KUKA KRL data list: tipdress2.dat

&ACCESS RV1
&REL 33
&COMMENT TIPDRESS EXTERNAL GUN 2
DEFDAT  TIPDRESS2
;FOLD EXTERNAL DECLARATIONS;%{PE}%MKUKATPBASIS,%CEXT,%VCOMMON,%P
;FOLD GRIPPERTECH EXT
EXT  H50 (INT  :IN,INT  :IN,INT  :IN,GRP_TYP  :IN )
;ENDFOLD (GRIPPERTECH EXT)
;FOLD SPOTTECH EXT
EXT  USERSPOT (S_COMMAND  :IN,SPOT_TYPE  :IN )
;ENDFOLD (SPOTTECH EXT)
;FOLD BASISTECH EXT;%{PE}%MKUKATPBASIS,%CEXT,%VEXT,%P
EXT  BAS (BAS_COMMAND  :IN,REAL  :IN )
DECL INT SUCCESS
;ENDFOLD (BASISTECH EXT)
;FOLD USER EXT;%{E}%MKUKATPUSER,%CEXT,%VEXT,%P
;Make here your modifications
;ENDFOLD (USER EXT)
;ENDFOLD (EXTERNAL DECLERATIONS)
;FOLD USER EXT;%{}%V2.2.2,%MKUKATPUSER,%CEXT,%VEXT,%P
;Make here your modifications
DECL BOOL TIPKONTROLE
DECL INT ANSWER
DECL INT WAITTIME=5
;ENDFOLD
;ENDFOLD
DECL INT I

;******************************
;*     E6POS Declarations     *
;******************************

DECL E6POS XP10={X 1812.73999,Y -758.109497,Z 1603.28101,A -10.9368095,B 87.2611084,C -2.35136199,S 6,T 50,E1 0.0,E2 0.0,E3 0.0,E4 0.0,E5 0.0,E6 0.0}
DECL E6POS XP20={X -1662.00305,Y -1200.49304,Z 238.679993,A 92.3594437,B 77.6989288,C -175.853195,S 6,T 26,E1 -667.745789,E2 0.0,E3 0.0,E4 0.0,E5 0.0,E6 0.0}
DECL E6POS XBEFORETIPDRESS={X -1664.84497,Y -1195.28101,Z 131.821106,A 92.7083206,B 79.2879791,C -177.241806,S 6,T 26,E1 -667.74939,E2 0.0,E3 0.0,E4 0.0,E5 0.0,E6 0.0}
DECL E6POS XDRESS_POS={X -1664.83301,Y -1250.33301,Z 131.817993,A 92.7068863,B 79.2882233,C -177.243393,S 6,T 26,E1 -667.74762,E2 0.0,E3 0.0,E4 0.0,E5 0.0,E6 0.0}
DECL E6POS XAFTERTIPDRESS={X -1664.84497,Y -1195.28101,Z 131.821106,A 92.7083206,B 79.2879791,C -177.241806,S 6,T 26,E1 -667.74939,E2 0.0,E3 0.0,E4 0.0,E5 0.0,E6 0.0}
DECL E6POS XBEST_PRACKTICE={X -1662.02905,Y -1184.83496,Z 277.771301,A 92.3578873,B 77.6946869,C -175.853302,S 6,T 26,E1 -667.74762,E2 0.0,E3 0.0,E4 0.0,E5 0.0,E6 0.0}
DECL E6POS XP30={X -958.122009,Y 929.273499,Z 985.610474,A 92.0788727,B 72.5539932,C -179.8358,S 6,T 26,E1 -2887.17505,E2 0.0,E3 0.0,E4 0.0,E5 0.0,E6 0.0}

;******************************
;*      FDAT Declarations     *
;******************************

DECL FDAT FP10={TOOL_NO 14,BASE_NO 0,IPO_FRAME #BASE,TQ_STATE FALSE}
DECL FDAT FP20={TOOL_NO 1,BASE_NO 0,IPO_FRAME #BASE}
DECL FDAT FBEFORETIPDRESS={TOOL_NO 1,BASE_NO 0,IPO_FRAME #BASE}
DECL FDAT FDRESS_POS={TOOL_NO 1,BASE_NO 0,IPO_FRAME #BASE}
DECL FDAT FAFTERTIPDRESS={TOOL_NO 1,BASE_NO 0,IPO_FRAME #BASE}
DECL FDAT FBEST_PRACKTICE={TOOL_NO 1,BASE_NO 0,IPO_FRAME #BASE}
DECL FDAT FP30={TOOL_NO 1,BASE_NO 0,IPO_FRAME #BASE}

;******************************
;*  PDAT & LDAT Declarations  *
;******************************

DECL PDAT PH={VEL 100.0,ACC 100.0,APO_DIST 100.0}

DECL E6POS XBEST_PRAKTISCH={X 1813.98499,Y -755.127197,Z 1603.28101,A -10.8495102,B 87.2611771,C -2.35826492,S 6,T 50,E1 0.0,E2 0.0,E3 0.0,E4 0.0,E5 0.0,E6 0.0}
DECL SPOT_SUGG_T LAST_SPOT={GUN[] "1                       ",RETR_CMD[] "#OPN                    ",CHOISE[] "#FIRST                  ",CLO_TM[] "0                       ",PGNO1[] "1                       ",PRESS1[] "0                       ",PGNO2[] "1                       ",PRESS2[] "0                       ",SPOT_PARAMS[] "SDAT3                   "}
DECL BASIS_SUGG_T LAST_BASIS={POINT1[] "Best_Praktisch          ",POINT2[] "Best_Praktisch          ",CP_PARAMS[] "CPDAT0                  ",PTP_PARAMS[] "H                       ",CONT[] "                        ",CP_VEL[] "2.0                     ",PTP_VEL[] "100                     ",SPL_NAME[] "S0                      "}
DECL FDAT FBest_Praktisch={TOOL_NO 14,BASE_NO 0,IPO_FRAME #BASE,POINT2[] " ",TQ_STATE FALSE}
DECL PDAT PPDAT1={VEL 100.0,ACC 100.0,APO_DIST 100.0}
DECL E6POS XBest_Praktice={X -1662.07202,Y -1184.76196,Z 277.795013,A 92.3631592,B 77.6921463,C -175.8461,S 6,T 26,E1 -667.74762,E2 0.0,E3 0.0,E4 0.0,E5 0.0,E6 0.0}
DECL FDAT FBest_Praktice={TOOL_NO 1,BASE_NO 0,IPO_FRAME #BASE,POINT2[] " "}
DECL E6POS XP21={X -929.55603,Y -159.533905,Z 748.283386,A 92.0804672,B 72.5703812,C -179.830597,S 6,T 26,E1 -2646.86792,E2 0.0,E3 0.0,E4 0.0,E5 0.0,E6 0.0}
DECL FDAT FP21={TOOL_NO 1,BASE_NO 0,IPO_FRAME #BASE}
DECL E6POS XP31={X -1185.09497,Y -662.41571,Z 415.422485,A 99.845192,B 75.8905869,C -168.599792,S 6,T 26,E1 -1294.38501,E2 0.0,E3 0.0,E4 0.0,E5 0.0,E6 0.0}
DECL FDAT FP31={TOOL_NO 1,BASE_NO 0,IPO_FRAME #BASE}
ENDDAT
